FUNCTION_BLOCK ASSEMBLE_AW_FROM_AQ (* this Function combines the 8 AQ (QUARTER) adapters to a AW (WORD) *)
  (* Standard: 61499-2; Description: Copyright (c) 2026 Meisterschulen am Ostbahnhof SPDX-License-Identifier: EPL-2.0 *)
  (* Version 1.0, 2026-05-16, Franz Höpfinger, Meisterschulen am Ostbahnhof, initial API and implementation and/or initial documentation *)
  PACKAGE adapter::assembling;
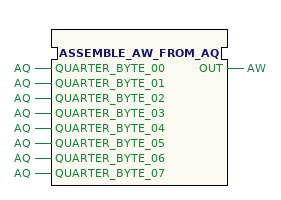
  SOCKETS
    QUARTER_BYTE_00 : adapter::types::unidirectional::AQ; (* Quarter 0 *)
    QUARTER_BYTE_01 : adapter::types::unidirectional::AQ; (* Quarter 1 *)
    QUARTER_BYTE_02 : adapter::types::unidirectional::AQ; (* Quarter 2 *)
    QUARTER_BYTE_03 : adapter::types::unidirectional::AQ; (* Quarter 3 *)
    QUARTER_BYTE_04 : adapter::types::unidirectional::AQ; (* Quarter 4 *)
    QUARTER_BYTE_05 : adapter::types::unidirectional::AQ; (* Quarter 5 *)
    QUARTER_BYTE_06 : adapter::types::unidirectional::AQ; (* Quarter 6 *)
    QUARTER_BYTE_07 : adapter::types::unidirectional::AQ; (* Quarter 7 *)
  END_SOCKETS
  PLUGS
    OUT : adapter::types::unidirectional::AW; (* WORD Output *)
  END_PLUGS
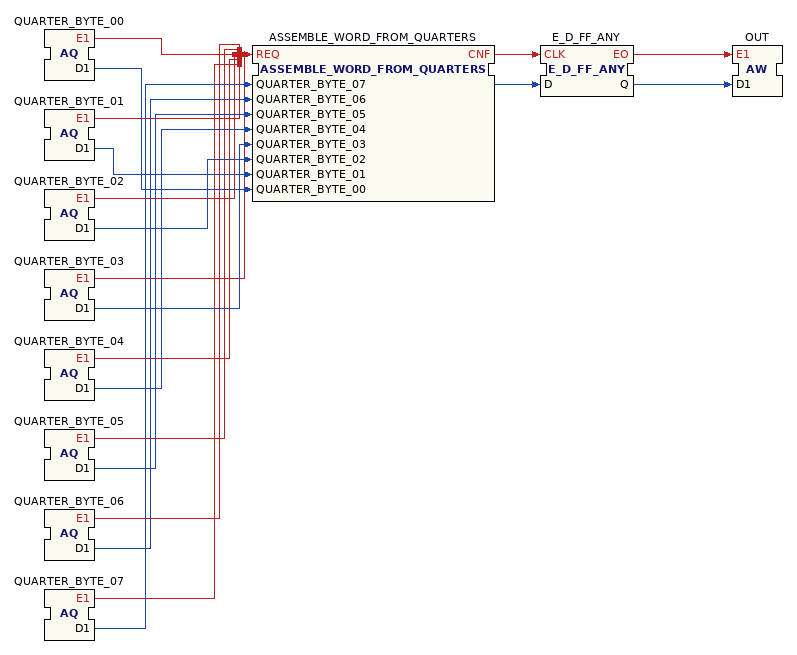
  FBS
    ASSEMBLE_WORD_FROM_QUARTERS : eclipse4diac::utils::assembling::ASSEMBLE_WORD_FROM_QUARTERS;
    E_D_FF_ANY : iec61499::events::E_D_FF_ANY;
  END_FBS
  EVENT_CONNECTIONS
    QUARTER_BYTE_00.E1 TO ASSEMBLE_WORD_FROM_QUARTERS.REQ;
    QUARTER_BYTE_01.E1 TO ASSEMBLE_WORD_FROM_QUARTERS.REQ;
    QUARTER_BYTE_02.E1 TO ASSEMBLE_WORD_FROM_QUARTERS.REQ;
    QUARTER_BYTE_03.E1 TO ASSEMBLE_WORD_FROM_QUARTERS.REQ;
    QUARTER_BYTE_04.E1 TO ASSEMBLE_WORD_FROM_QUARTERS.REQ;
    QUARTER_BYTE_05.E1 TO ASSEMBLE_WORD_FROM_QUARTERS.REQ;
    QUARTER_BYTE_06.E1 TO ASSEMBLE_WORD_FROM_QUARTERS.REQ;
    QUARTER_BYTE_07.E1 TO ASSEMBLE_WORD_FROM_QUARTERS.REQ;
    ASSEMBLE_WORD_FROM_QUARTERS.CNF TO E_D_FF_ANY.CLK;
    E_D_FF_ANY.EO TO OUT.E1;
  END_CONNECTIONS
  DATA_CONNECTIONS
    ASSEMBLE_WORD_FROM_QUARTERS. TO E_D_FF_ANY.D;
    E_D_FF_ANY.Q TO OUT.D1;
    QUARTER_BYTE_07.D1 TO ASSEMBLE_WORD_FROM_QUARTERS.QUARTER_BYTE_07;
    QUARTER_BYTE_06.D1 TO ASSEMBLE_WORD_FROM_QUARTERS.QUARTER_BYTE_06;
    QUARTER_BYTE_05.D1 TO ASSEMBLE_WORD_FROM_QUARTERS.QUARTER_BYTE_05;
    QUARTER_BYTE_04.D1 TO ASSEMBLE_WORD_FROM_QUARTERS.QUARTER_BYTE_04;
    QUARTER_BYTE_03.D1 TO ASSEMBLE_WORD_FROM_QUARTERS.QUARTER_BYTE_03;
    QUARTER_BYTE_02.D1 TO ASSEMBLE_WORD_FROM_QUARTERS.QUARTER_BYTE_02;
    QUARTER_BYTE_01.D1 TO ASSEMBLE_WORD_FROM_QUARTERS.QUARTER_BYTE_01;
    QUARTER_BYTE_00.D1 TO ASSEMBLE_WORD_FROM_QUARTERS.QUARTER_BYTE_00;
  END_CONNECTIONS
END_FUNCTION_BLOCK
